FUNCTION_BLOCK Generator
  (* Standard: 61499-2 *)
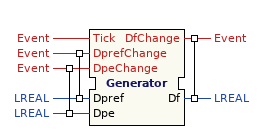
  EVENT_INPUT
    Tick;
    DprefChange WITH Dpref;
    DpeChange WITH Dpe;
  END_EVENT
  EVENT_OUTPUT
    DfChange WITH Df;
  END_EVENT
  VAR_INPUT
    Dpref : LREAL;
    Dpe : LREAL := 0.1;
  END_VAR
  VAR_OUTPUT
    Df : LREAL;
  END_VAR
  VAR
    StepSize : LREAL := 0.1;
    Kp : LREAL := 120;
    Tp : LREAL := 20;
    R : LREAL := 2.4;
  END_VAR
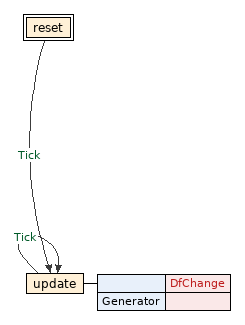
  EC_STATES
    reset;
    update : -> DfChange, Generator;
  END_STATES
  EC_TRANSITIONS
    reset TO update := Tick;
    update TO update := Tick;
  END_TRANSITIONS
  ALGORITHM Generator IN ST:
        Df := Df + ((Kp * Dpref - (Kp / R + 1) * Df - Kp * (Dpe)) / Tp) * StepSize;
  END_ALGORITHM
END_FUNCTION_BLOCK
